FUNCTION CalculateAverage : REAL
VAR_INPUT
	 aWeight : ARRAY[1..20] OF REAL;
END_VAR
VAR
	 i : INT;
    rSum : REAL := 0;
	nValidCount : INT := 0;
	iValidCount: INT;
END_VAR

FOR i := 1 TO 20 DO
	 IF (aWeight[i] >=50.0) AND (aWeight[i] <= 500.0) THEN
         rSum := rSum + aWeight[i];
		 iValidCount := iValidCount + 1;
    END_IF
END_FOR


IF iValidCount > 0 THEN
    CalculateAverage := rSum / iValidCount;
ELSE
    CalculateAverage := 0.0;   
END_IF

END_FUNCTION

(* stored: Version 1.1.0.1, ProductVersion 3.1.4024.16
   POU CalculateAverage: Id {dcc3e047-7d3e-4918-9fd2-626449e2c964}, SpecialFunc None *)
